// TIA Portal V19 export
TYPE "LubrMotorPump_HMI"
// stored: Access Published
   STRUCT
      Alarm : Bool;
      Running : Bool;
   END_STRUCT;
END_TYPE
